(* IEC 61131-3 sources: ICSQuartz/benchmarks/oscat_basic_trime/src, 1 file *)

(* ---- program.st ---- *)
PROGRAM PLC_PRG
VAR_INPUT
    in_STR: STRING;
END_VAR

TRIME(in_STR);

END_PROGRAM
